# EPICS StreamDevice protocol: streamdeviceApp/Db/danfysik.proto
# StreamDevice Protocol for Danfysik System SYS8X00 Power Supply
# Based on Danfysik System SYS8X00 Command Reference
# Created: January 2026
#
# NOTE: All commands require addressing the power supply first with ADR command
# The ADDR parameter must be passed from the database records

# Communication parameters
terminator   = CR;          # Commands terminated by Carriage Return
replyterminator = CR;    # Responses terminated by Line Feed + Carriage Return
replytimeout = 2000;        # 2 second timeout for responses
readtimeout  = 2000;        # 2 second read timeout
extrainput   = Ignore;      # Ignore extra input

# Error handling - responses with error include "?BELL" (ASCII 7)
# We'll handle this by checking for the bell character in responses

################################################################################
# Basic Control Commands
################################################################################

# Power ON - Switch main power contactor ON
power_on    { out "ADR \$1"; out "N"; }

# Power OFF - Switch main power contactor OFF
power_off   { out "ADR \$1"; out "F"; }

# Global OFF - Soft shutdown ensuring DAC at minimum before turning off
global_off  { out "ADR \$1"; out "GOFF"; }

# Reset interlocks - Clear latched error states
reset       { out "ADR \$1"; out "RS"; }

################################################################################
# Remote/Local Control
################################################################################

# Switch to remote control
remote_ctrl { out "ADR \$1"; out "REM"; }

# Switch to local control
local_ctrl  { out "ADR \$1"; out "LOC"; }

# Read current control mode
get_cmd_mode { out "ADR \$1"; out "CMD"; in "%3c"; }

# Read detailed control state
get_cmd_state { out "ADR \$1"; out "CMDSTATE"; in "%8c"; }

# Remote lock - prevent local panel from taking control
remote_lock { out "ADR \$1"; out "RLOCK"; }

# Unlock from remote (emergency use)
unlock      { out "ADR \$1"; out "UNLOCK"; }

################################################################################
# Addressing Commands
################################################################################

# Read MPS address
get_address { out "ADR"; in "%d"; }

# Set MPS address (00-63)
set_address { out "ADR \$1"; out "ADR %02d"; }

# Listen all mode - for multi-unit configuration
listen_all  { out "LALL"; }

################################################################################
# Current Setting and Reading (DAC based)
################################################################################

# Write current setpoint (6 digits: 000000-999999)
# Formula: DAC_value = (Desired_Current / Nominal_Current) * 1,000,000
set_current { out "ADR \$1"; out "WA %06d"; }

# Read current setpoint (6 digits)
# Formula: Current = Nominal_Current * (DAC_value / 1,000,000)
get_current_sp { out "ADR \$1"; out "RA"; in "%d"; }

# Write ramp end value (for ramping)
set_ramp_end { out "ADR \$1"; out "WAR %06d"; }

# Read ramp end value
get_ramp_end { out "ADR \$1"; out "RAR"; in "%d"; }

################################################################################
# Ramp Speed Control
################################################################################

# Write ramp speed (001-100 = 0.1% to 10% of rated current per second)
set_ramp_speed { out "ADR \$1"; out "WR %03d"; }

# Read ramp speed
get_ramp_speed { out "ADR \$1"; out "RR"; in "%d"; }

################################################################################
# ADC Channel Readings
################################################################################

# Read output current (Channel 0) - returns (I/In)*100
get_output_current { out "ADR \$1"; out "AD 0"; in "%d"; }

# Read Tesla field (Channel 1) - returns T*100
get_tesla { out "ADR \$1"; out "AD 1"; in "%d"; }

# Read output voltage (Channel 2) - returns (V/Vn)*100
get_output_voltage { out "ADR \$1"; out "AD 2"; in "%d"; }

# Read +15V supply (Channel 3) - returns V*10
get_p15v { out "ADR \$1"; out "AD 3"; in "%d"; }

# Read -15V supply (Channel 4) - returns V*10
get_m15v { out "ADR \$1"; out "AD 4"; in "%d"; }

# Read +5V supply (Channel 5) - returns V*10
get_p5v { out "ADR \$1"; out "AD 5"; in "%d"; }

# Read delta temperature (Channel 6) - returns Deg.C*10 with sign
get_temp_delta { out "ADR \$1"; out "AD 6"; in "%d"; }

# Read transistor bank Vce (Channel 7) - returns V
get_vce { out "ADR \$1"; out "AD 7"; in "%d"; }

# Read optional high-res current (Channel 8) - returns (I/In)*100000 if equipped
get_hires_current { out "ADR \$1"; out "AD 8"; in "%d"; }

# Read aux current (Channel 9) - returns (I/In)*120
get_aux_current { out "ADR \$1"; out "AD 9"; in "%d"; }

################################################################################
# Polarity Control
################################################################################

# Read polarity status
get_polarity { out "ADR \$1"; out "PO"; in "%c"; }

# Set normal polarity
set_pol_normal { out "ADR \$1"; out "PO+"; }

# Set reverse polarity
set_pol_reverse { out "ADR \$1"; out "PO-"; }

################################################################################
# Status and Error Monitoring
################################################################################

# Read 24-bit status string (interlocks, polarity, on/off status)
# Returns 24 characters: '!' = error/non-normal, '.' = normal
get_status { out "ADR \$1"; out "S1"; in "%24c"; }

# Read the same 24-character status string, but decoded as a single 24-bit
# mask (character 1 = bit 23 .. character 24 = bit 0) using StreamDevice's
# binary converter, so individual bits can be extracted with calc records.
get_status_bits { out "ADR \$1"; out "S1"; in "%24B.!"; }

################################################################################
# Communication Control
################################################################################

# Set error response mode to text
error_text { out "ADR \$1"; out "ERRT"; }

# Set error response mode to codes
error_code { out "ADR \$1"; out "ERRC"; }

# Suppress detailed error messages (only BELL on error)
no_error { out "ADR \$1"; out "NERR"; }

# Auto-answer mode for certain commands
answer_mode { out "ADR \$1"; out "ASW"; }

# Disable auto-answer mode
no_answer { out "ADR \$1"; out "NASW"; }

# Set baud rate (19200, 9600, 4800, 2400, 1200, 600, 300, 150)
set_baud { out "ADR \$1"; out "BAUD %d"; }

################################################################################
# Information Commands
################################################################################

# Read unit information (serial number, type)
get_info { out "ADR \$1"; out "PRINT"; in "%80c"; }

# Read firmware version information
# Reply starts with a blank line (bare CR) before the actual text line,
# so the first "in" consumes and discards it.
get_version { out "ADR \$1"; out "VER"; in ""; in "%80c"; }

################################################################################
# Binary Quick Read Commands (for high-speed monitoring)
################################################################################

# Quick binary read of high-definition current ADC (24-bit raw)
# Note: StreamDevice may need special handling for binary data
quick_current_bin { out "ADR \$1"; out "?1"; in "%4r"; }

# Quick binary read of status (32-bit)
quick_status_bin { out "ADR \$1"; out "?2"; in "%4r"; }

# Quick binary read combined status + ADC (32-bit + 24-bit)
quick_combined_bin { out "ADR \$1"; out "?3"; in "%7r"; }

# Read ADC 100% calibration value (24-bit)
quick_cal_bin { out "ADR \$1"; out "?4"; in "%4r"; }

################################################################################
# Sequence Control
################################################################################

# Trigger programmed sequence from first position (stack 0-3)
trigger_seq { out "ADR \$1"; out "TS %d"; }

################################################################################
# Synchronization
################################################################################

# Synchronize communication (equivalent to Ctrl+V, ASCII 16)
# Note: This may need special handling in StreamDevice
sync_comm { out "\x10"; wait 150; out "\r"; }

################################################################################
# Composite Operations for Common Use Cases
################################################################################

# Initialize power supply for remote operation
init_remote {
    out "ADR \$1";       # Address the power supply
    out "REM";           # Switch to remote
    out "ERRT";          # Enable text error messages
    out "RS";            # Clear any latched errors
}

# Safe shutdown sequence
safe_shutdown {
    out "ADR \$1";       # Address the power supply
    out "GOFF";          # Global off (soft shutdown)
}

# Read all vital parameters in sequence
read_all_params {
    out "ADR \$1";               # Address the power supply
    out "RA"; in "%d";           # Current setpoint
    out "AD 0"; in "%d";         # Output current
    out "AD 2"; in "%d";         # Output voltage
    out "PO"; in "%c";           # Polarity
    out "S1"; in "%24c";         # Status
    out "CMD"; in "%3c";         # Control mode
}

################################################################################
# Error handling with status check
################################################################################

# Set current with status verification
set_current_safe {
    out "ADR \$1";              # Address the power supply
    out "WA %06d";              # Set current
    out "S1"; in "%24c";        # Check status after
}

# Power on with status check
power_on_safe {
    out "ADR \$1";              # Address the power supply
    out "N";                    # Power on
    out "S1"; in "%24c";        # Check status
}
